{attribute 'GeneratedUsingTerminal: EL3681-0000-0018'}
{attribute addProperty BoxType "EL3681-0000-0018"}
{attribute addProperty Id "UnderrangeBOOL1OverrangeBOOL1Extended_rangeBOOL1Data_invalidBOOL1Range_invalidBOOL1Autorange_disabledBOOL1ErrorBOOL1Calibration_in_progressBOOL1TxPDO_StateBOOL1TxPDO_ToggleBOOL1"}
{attribute addProperty CRC "1374726436"}
{attribute addProperty Size "10"}
TYPE Status_51F0A924 :
STRUCT
	{attribute addProperty Name "Underrange"}
	Underrange : BOOL;
	{attribute addProperty Name "Overrange"}
	Overrange : BOOL;
	{attribute addProperty Name "Extended_range"}
	Extended_range : BOOL;
	{attribute addProperty Name "Data_invalid"}
	Data_invalid : BOOL;
	{attribute addProperty Name "Range_invalid"}
	Range_invalid : BOOL;
	{attribute addProperty Name "Autorange_disabled"}
	Autorange_disabled : BOOL;
	{attribute addProperty Name "Error"}
	Error : BOOL;
	{attribute addProperty Name "Calibration_in_progress"}
	Calibration_in_progress : BOOL;
	{attribute addProperty Name "TxPDO_State"}
	TxPDO_State : BOOL;
	{attribute addProperty Name "TxPDO_Toggle"}
	TxPDO_Toggle : BOOL;
END_STRUCT
END_TYPE

(* stored: Version 1.2.0.0, ProductVersion 3.1.4024.9
   DUT Status_51F0A924: Id {6988e327-dd14-4c8f-a85c-3e9879ed97ac} *)
